Fanuc TP program (LS listing): IONCE.LS

/PROG  IONCE	  Cond
/ATTR
OWNER		= MNEDITOR;
COMMENT		= "iOnce";
PROG_SIZE	= 0;
CREATE		= DATE 26-01-01  TIME 00:00:00;
MODIFIED	= DATE 26-01-01  TIME 00:00:00;
FILE_NAME	= ;
VERSION		= 0;
LINE_COUNT	= 1;
MEMORY_SIZE	= 0;
PROTECT		= READ_WRITE;
TCD:  STACK_SIZE	= 0,
      TASK_PRIORITY	= 50,
      TIME_SLICE	= 0,
      BUSY_LAMP_OFF	= 0,
      ABORT_REQUEST	= 0,
      PAUSE_REQUEST	= 0;
DEFAULT_GROUP	= *,*,*,*,*;
CONTROL_CODE	= 00000000 00000000;
/MN
   1:  WHEN DO[2]=ON+,CALL TONCE ;
/POS
/END
